KUKA KRL program: Cordon_vertical.src, Cordon_vertical.dat

--- Cordon_vertical.src ---
&ACCESS RVO1
&COMMENT
DEF Cordon_vertical ( )
; Programa desarrollado por Mauricio Sol�s para pruebas de soldadura en el CIMA.

DECL REAL dx, dy, dz, r_speed
DECL E6POS p0_rel

;FOLD INI
  ;FOLD BASISTECH INI
    GLOBAL INTERRUPT DECL 3 WHEN $STOPMESS==TRUE DO IR_STOPM ( )
    INTERRUPT ON 3
    BAS (#INITMOV,0 )
  ;ENDFOLD (BASISTECH INI)
  ;FOLD USER INI
    ;Make your modifications here

  ;ENDFOLD (USER INI)
;ENDFOLD (INI)

; PTP p0 Vel= 100 % PDAT1 Tool[5]:torcha_metalurgia Base[0]
;FOLD PTP p0  Vel=100 % PDAT1 Tool[5] Base[1];%{PE}%R 5.6.11,%MKUKATPBASIS,%CMOVE,%VPTP,%P 1:PTP, 2:p0, 3:, 5:100, 7:PDAT1
$BWDSTART=FALSE
PDAT_ACT=PPDAT1
FDAT_ACT=Fp0
BAS(#PTP_PARAMS,100)
PTP Xp0
;ENDFOLD

p0_rel = Xp0; Punto inicial (inicio del cord�n) a 12 mm de la superficie,
; para dar espacio al cord�n de soldadura.
; Este es el �nico punto que se le ense�a al robot (touch up).

r_speed = 0.005; Velocidad de avance (m/s)

; Desfases aplicados al punto inicial, utilzar si se requiere un nuevo cord�n a
; cierta distancia de los ya realizados.
dx = 0
dy = 0
dz = 0

p0_rel.x = Xp0.x + dx
p0_rel.y = Xp0.y + dy
p0_rel.z = Xp0.z + dz

;PTP p0_rel

HALT ;Detener justo antes de comenzar la soldadura para que el operador de la
; se�al de partida.

cordon_vert(p0_rel, 80, r_speed, 2, 1)

END

; En esta funci�n, para cada cord�n, se realiza un trayecto de ida y otro de
; vuelta. Lo que equivale en la pr�ctica a dos cordones por cada cord�n
; pasado como argumento en num_cor.
DEF cordon_vert(origen:IN, len:IN, speed:IN, dz:IN, num_cor:IN)
  DECL E6POS origen
  DECL REAL len
  DECL REAL speed
  DECL REAL dz
  DECL INT num_cor

  DECL E6POS final
  DECL E6POS ori, ori_up
  DECL E6POS fin, fin_up
  DECL INT N

  ori_up.z = ori_up.z + 150; Altura de seguridad para que la torcha se mueva
  ; horizontalmente sin obst�culos.
  fin.y = fin.y - len; Cambiar el signo de la operaci�n para realizar el cord�n
  ; en el sentido opuesto.
  fin_up = fin
  fin_up.z = fin_up.z + 150
  final = fin

  FOR N = 0 TO num_cor
    ori.z = origen.z + 2*N * dz
    fin.z = final.z + 2*N * dz

    BAS(#VEL_CP, 0.2); Ajustar velocidad de desplazamiento (m/s).
    PTP ori_up
    LIN ori

    BAS(#VEL_CP, speed); Ajustar velocidad de avance durante la soldadura (m/s).
    $OUT[40] = TRUE; Enciende soldadora.

    WAIT Time= 0.8 sec
    LIN fin
    $OUT[40] = FALSE; Apaga soldadora.

    BAS(#VEL_CP, 0.2)
    LIN fin_up
    HALT; Espera se�al del operador para continuar. Aqu� se verifica con pistola
    ; de temperatura que esta haya bajado de 100 �C aprox. para continuar con el
    ; siguiente cord�n.
    ; En la pr�ctica, nosotros detuvimos el programa ac�, cambiamos el offset
    ; con dx, dy, dz, y comenzamos de nuevo.

    ; Eleva torcha para realizar cord�n de vuelta sobre el anterior.
    ori.z = origen.z + (2*N + 1) * dz
    fin.z = final.z + (2*N + 1) * dz

    LIN fin
    BAS(#VEL_CP, speed)
    $OUT[40] = TRUE
    WAIT Time= 0.8 sec
    LIN ori
    $OUT[40] = FALSE

    BAS(#VEL_CP, 0.2)
    LIN ori_up
    HALT

  ENDFOR

END

--- Cordon_vertical.dat ---
&ACCESS RVO1
&COMMENT
DEFDAT Cordon_vertical PUBLIC
;FOLD EXTERNAL DECLARATIONS;%{PE}%MKUKATPBASIS,%CEXT,%VCOMMON,%P
;FOLD BASISTECH EXT;%{PE}%MKUKATPBASIS,%CEXT,%VEXT,%P
EXT  BAS (BAS_COMMAND  :IN,REAL  :IN )
DECL INT SUCCESS
;ENDFOLD (BASISTECH EXT)
;FOLD USER EXT;%{E}%MKUKATPUSER,%CEXT,%VEXT,%P
;Make here your modifications

;ENDFOLD (USER EXT)
;ENDFOLD (EXTERNAL DECLERATIONS)
DECL BASIS_SUGG_T LAST_BASIS={POINT1[] "P0",POINT2[] "P0",CP_PARAMS[] "CPDAT0",PTP_PARAMS[] "PDAT1",CONT[] " ",CP_VEL[] "2",PTP_VEL[] "100",SYNC_PARAMS[] " ",SPL_NAME[] " "}
DECL E6POS XP0={X 0.0,Y 0.0,Z 0.0,A 0.0,B 0.0,C 0.0,S 0,T 0,E1 0.0,E2 0.0,E3 0.0,E4 0.0,E5 0.0,E6 0.0}
DECL FDAT FP0={TOOL_NO 5,BASE_NO 1,IPO_FRAME #BASE,POINT2[] " ",TQ_STATE FALSE}
DECL PDAT PPDAT1={VEL 100,ACC 100,APO_DIST 100}
ENDDAT
